TYPE ST_ContentOUT1 :
STRUCT
	DefaultIdentity   :ST_DefaultIdentityOUT1;
	ExpectedItemCount	:STRING;
	ItemReadRate		:STRING;
	ItemList			:ST_ItemListOUT1;
END_STRUCT
END_TYPE

(* stored: Version 1.1.0.1, ProductVersion 3.1.4024.13
   DUT ST_ContentOUT1: Id {37236852-75be-4648-8f2c-985d27fbf25f} *)
